{attribute 'qualified_only'}
{attribute 'strict'}
{attribute 'to_string'}
TYPE eState :
(
	None 			:= 0,
	Finalized:= 1,
	Unconfigured 	:= 2,
	ErrorProcessing:= 3,
	CleaningUp:= 4,
	ShuttingDown:= 5,	
	Configuring := 6,			
	Inactive := 7,			
	Deactivating := 8,	
	Activating 	:= 9,		
	Active:= 10
);
END_TYPE

(* stored: Version 1.1.0.1, ProductVersion 3.1.4026.18
   DUT eState: Id {a1b2c3d4-1111-1111-1111-111111111111} *)
